PROGRAM SFC_Test
VAR
	Step0:SFCStepType;
	Step1:SFCStepType;
	Step2:SFCStepType;
	Step3:SFCStepType;
	Step4:SFCStepType;
	Switch1:BOOL;
	Switch2:BOOL;
	Lamp1:BOOL;
	Lamp2:BOOL;
	Lamp3:BOOL;
	Counter:INT;
	Step0_Counter:INT;
	Step1_Counter:INT;
	
END_VAR

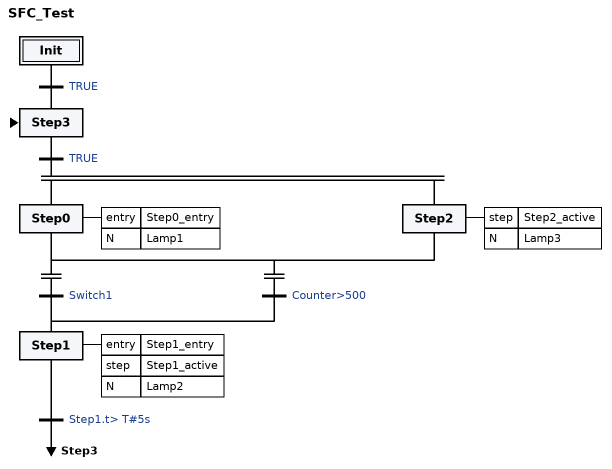
INITIAL_STEP Init:
END_STEP
TRANSITION FROM Init TO Step3
    := TRUE;
END_TRANSITION
STEP Step3:
END_STEP
TRANSITION FROM Step3 TO (Step0, Step2)
    := TRUE;
END_TRANSITION
STEP Step0:
    Step0_entry(P1);  // entry action
    Lamp1(N);
END_STEP
STEP Step2:
    Step2_active(N);  // step action
    Lamp3(N);
END_STEP
TRANSITION FROM (Step0, Step2) TO Step1
    := Switch1;
END_TRANSITION
TRANSITION FROM (Step0, Step2) TO Step1
    := Counter>500;
END_TRANSITION
STEP Step1:
    Step1_entry(P1);  // entry action
    Step1_active(N);  // step action
    Lamp2(N);
END_STEP
TRANSITION FROM Step1 TO Step3
    := Step1.t> T#5s;
END_TRANSITION

ACTION Step0_entry:
Step0_Counter:=500;
END_ACTION

ACTION Step1_active:
Step1_Counter:=Step1_Counter+1;
END_ACTION

ACTION Step1_entry:
Step1_Counter:=0;
Counter:=0;
END_ACTION

ACTION Step2_active:
Counter:=Counter+1;
END_ACTION

ACTION Step4_active:
;
END_ACTION

END_PROGRAM

(* stored: Version 1.1.0.1, ProductVersion 3.1.4022.10
   POU SFC_Test: Id {bfe15231-0978-40d1-b104-683ff9823199}, SpecialFunc None
   Action Step0_entry: Id {e9620b15-4c4a-465d-82b8-6b1b517525c8}
   Action Step1_active: Id {e9ed5433-5f5d-482d-a9a1-26b50c519575}
   Action Step1_entry: Id {b9a60d50-6371-4e08-ac9e-31b252a51eb7}
   Action Step2_active: Id {02981a39-af78-4f43-913f-5874ce7eac8a}
   Action Step4_active: Id {07904fef-ce70-4f30-9df6-87abe9da587a} *)
